Omron Sysmac Studio project TestingWithEuchnerCIPSafetySW (Sysmac Studio 1.54.0.64019, StandardProject)

# Controller PLC01: NX102-9000 version 1.60
Task PrimaryTask (priority 4, period or condition 2000): Program0

VAR_GLOBAL
    DataFromEagle : ARRAY[0..9] OF int;  (* network input *)
    DataToEagle : ARRAY[0..9] OF int;  (* network output *)
END_VAR

(* Program Program0: safety or other program stored in binary form, left out *)

PROGRAM Program0
VAR
    sw1 : BOOL;
    sw2 : BOOL;
END_VAR

(* Section Section0: ladder, written here as Structured Text *)

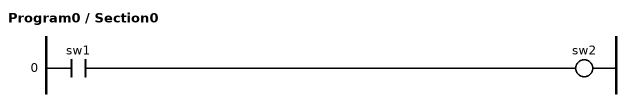
(* Rung 0 *)
sw2 := sw1;
END_PROGRAM